// SIMATIC S7-200 project (STEP 7-Micro/WIN), CPU 221 REL 01.10

SYMBOL_TABLE USER1
phim2            I0.2
phim4            I0.3
phim6            I0.4
phim8            I0.5
clear            I0.6
start            I0.0
stopp            I0.1
Den              Q0.0
END_SYMBOL_TABLE

ORGANIZATION_BLOCK MAIN:OB1
TITLE=
BEGIN
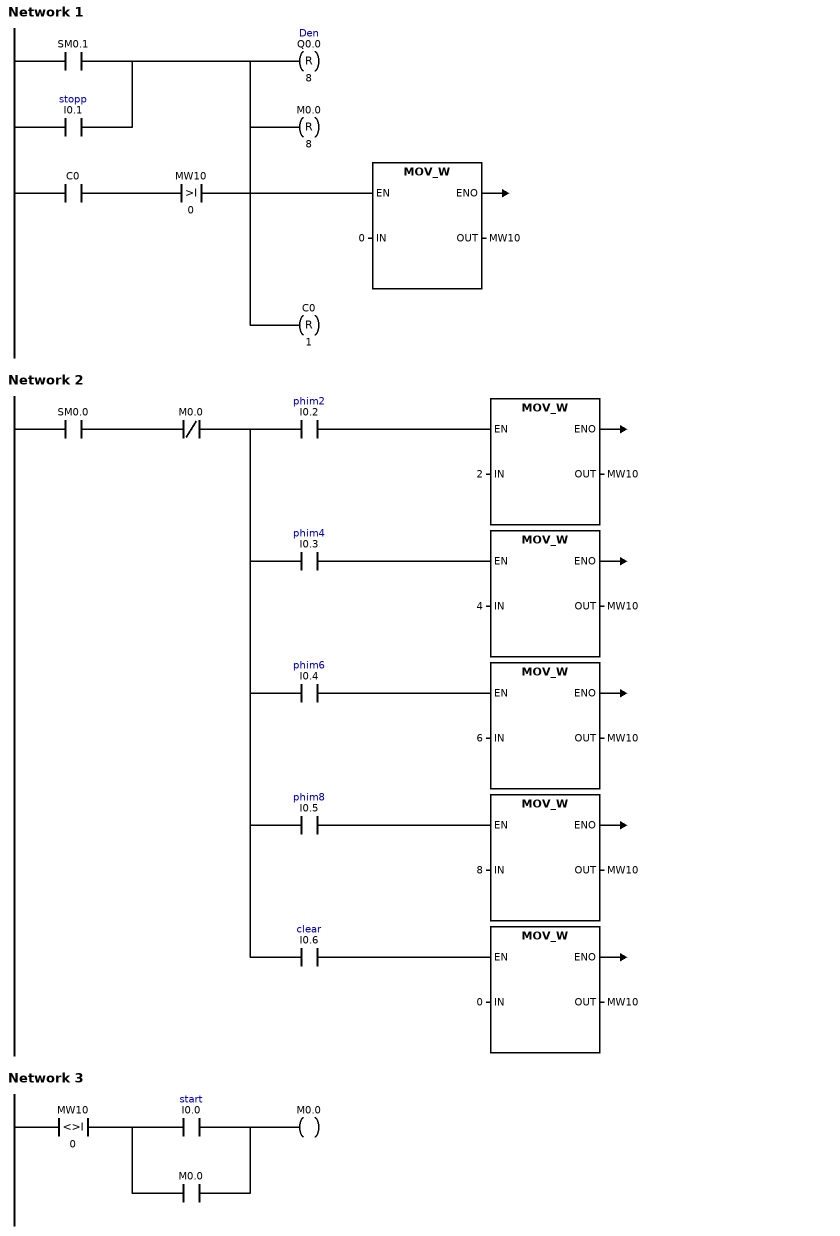
Network 1
LD     SM0.1
O      stopp:I0.1
LD     C0
AW>    MW10, 0
OLD
R      Den:Q0.0, 8
R      M0.0, 8
MOVW   0, MW10
R      C0, 1
Network 2
LD     SM0.0
AN     M0.0
LPS
A      phim2:I0.2
MOVW   2, MW10
LRD
A      phim4:I0.3
MOVW   4, MW10
LRD
A      phim6:I0.4
MOVW   6, MW10
LRD
A      phim8:I0.5
MOVW   8, MW10
LPP
A      clear:I0.6
MOVW   0, MW10
Network 3
LDW<>  MW10, 0
LD     start:I0.0
O      M0.0
ALD
=      M0.0
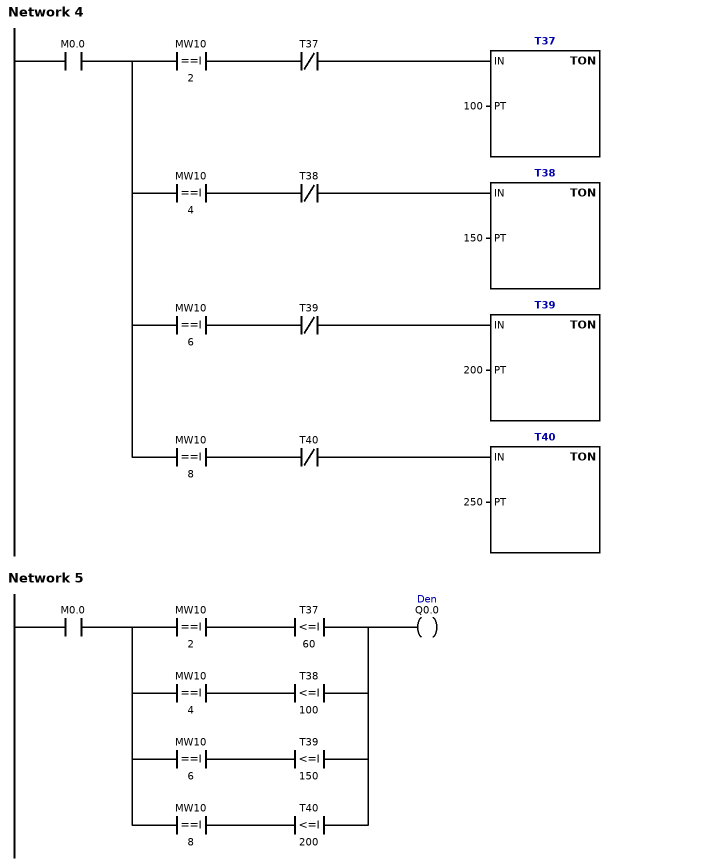
Network 4
LD     M0.0
LPS
AW=    MW10, 2
AN     T37
TON    T37, 100
LRD
AW=    MW10, 4
AN     T38
TON    T38, 150
LRD
AW=    MW10, 6
AN     T39
TON    T39, 200
LPP
AW=    MW10, 8
AN     T40
TON    T40, 250
Network 5
LD     M0.0
LDW=   MW10, 2
AW<=   T37, 60
LDW=   MW10, 4
AW<=   T38, 100
OLD
LDW=   MW10, 6
AW<=   T39, 150
OLD
LDW=   MW10, 8
AW<=   T40, 200
OLD
ALD
=      Den:Q0.0
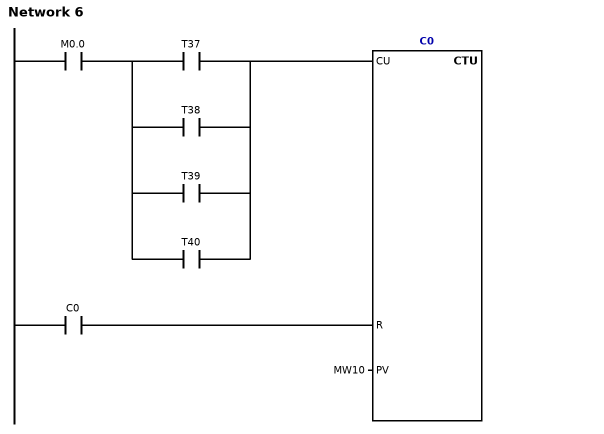
Network 6
LD     M0.0
LD     T37
O      T38
O      T39
O      T40
ALD
LD     C0
CTU    C0, MW10
END_ORGANIZATION_BLOCK
